(* IEC 61131-3 sources: openplc-validation-lab/plc_projects/runtime_smoke_test/pous/programs, 1 file *)

(* ---- main.st ---- *)
PROGRAM main
  VAR
    cycle_counter : DINT := 0;
    mb_command : UINT AT %MW0 := 0;
    mb_response : UINT AT %MW1 := 0;
    remote_hr0 : UINT AT %IW0 := 0;
  END_VAR

cycle_counter := cycle_counter + 1;
mb_response := mb_command + 1;

END_PROGRAM
